// TIA Portal V18 export
FUNCTION "IOT_DATA_FC" : Void   // FC1001, LAD
{ S7_Optimized_Access := 'TRUE' }
VERSION : 0.1
// stored: AutoNumber false, IsIECCheckEnabled true, SetENOAutomatically true, UDAEnableTagReadback false
BEGIN

REGION Network 1 (SCL)
   "IOT_DATA"."pump A Inlet" := "pressure"."pump A Inlet";
   "IOT_DATA"."pump B Inlet" := "pressure"."pump B Inlet";
   "IOT_DATA"."pump A Outlet" := "pressure"."pump A Outlet";
   "IOT_DATA"."pump B Outlet" := "pressure"."pump B Outlet";
END_REGION
END_FUNCTION
